SYSTEM Scenario_3
  (* Version 1.0, 2025-08-24, DEVIASH *)
  APPLICATION Scenario_3App (* VDMA *)
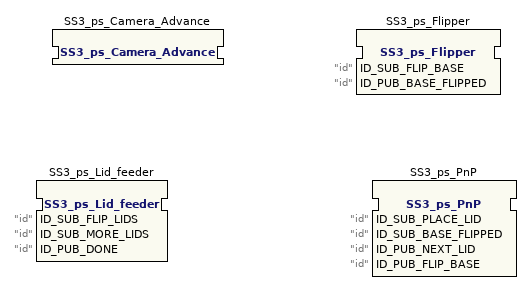
    (* Group S3_Capping_Station: Puting cap on the spinner *)
    FBS
      SS3_ps_Flipper : SS3_ps_Flipper(ID_SUB_FLIP_BASE := "id", ID_PUB_BASE_FLIPPED := "id"); {SET_ATTRIBUTE(GroupName, S3_Capping_Station)}
      SS3_ps_Lid_feeder : SS3_ps_Lid_feeder(ID_SUB_FLIP_LIDS := "id", ID_SUB_MORE_LIDS := "id", ID_PUB_DONE := "id"); {SET_ATTRIBUTE(GroupName, S3_Capping_Station)}
      SS3_ps_PnP : SS3_ps_PnP(ID_SUB_PLACE_LID := "id", ID_SUB_BASE_FLIPPED := "id", ID_PUB_NEXT_LID := "id", ID_PUB_FLIP_BASE := "id"); {SET_ATTRIBUTE(GroupName, S3_Capping_Station)}
      SS3_ps_Camera_Advance : SS3_ps_Camera_Advance; {SET_ATTRIBUTE(GroupName, S3_Capping_Station)}
    END_FBS
  END_APPLICATION
  APPLICATION Scenario_3_PreApp (* VDMA *)
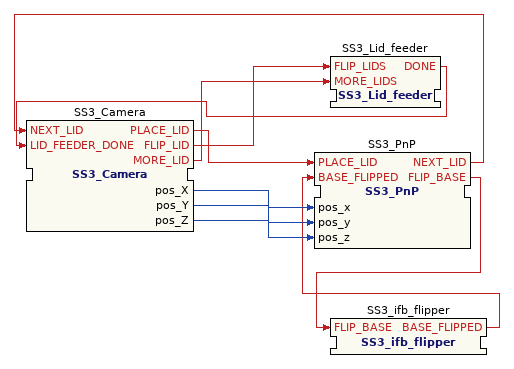
    (* Group S3_Capping_Station: Puting cap on the spinner *)
    FBS
      SS3_Lid_feeder : SS3_Lid_feeder; {SET_ATTRIBUTE(GroupName, S3_Capping_Station)}
      SS3_PnP : SS3_PnP; {SET_ATTRIBUTE(GroupName, S3_Capping_Station)}
      SS3_Camera : SS3_Camera; {SET_ATTRIBUTE(GroupName, S3_Capping_Station)}
      SS3_ifb_flipper : SS3_ifb_flipper; {SET_ATTRIBUTE(GroupName, S3_Capping_Station)}
    END_FBS
    EVENT_CONNECTIONS
      SS3_Camera.PLACE_LID TO SS3_PnP.PLACE_LID;
      SS3_PnP.NEXT_LID TO SS3_Camera.NEXT_LID;
      SS3_Camera.FLIP_LID TO SS3_Lid_feeder.FLIP_LIDS;
      SS3_Camera.MORE_LID TO SS3_Lid_feeder.MORE_LIDS;
      SS3_Lid_feeder.DONE TO SS3_Camera.LID_FEEDER_DONE;
      SS3_PnP.FLIP_BASE TO SS3_ifb_flipper.FLIP_BASE;
      SS3_ifb_flipper.BASE_FLIPPED TO SS3_PnP.BASE_FLIPPED;
    END_CONNECTIONS
    DATA_CONNECTIONS
      SS3_Camera.pos_X TO SS3_PnP.pos_x;
      SS3_Camera.pos_Y TO SS3_PnP.pos_y;
      SS3_Camera.pos_Z TO SS3_PnP.pos_z;
    END_CONNECTIONS
  END_APPLICATION
END_SYSTEM
